TYPE CTR_SIGNALS_INTERNAL :
STRUCT
	//motion control signals
	Enable					:BOOL;
	Execute_SPOS			:BOOL;
	Execute_MABS			:BOOL;
	Execute_MREL			:BOOL;
	Execute_RES				:BOOL;
	//Execute_VEL				:BOOL;
	Execute_HALT			:BOOL;
	Execute_STOP			:BOOL;
	Execute_HOME			:BOOL;	
	JogFw					:BOOL;
	JogBw					:BOOL;
	JogMode					:E_JogMode;
	SetLocation				:LREAL;
	SetPosition				:LREAL;
	SetVelocity				:LREAL;
	SetAccel				:LREAL;
	LimPos					:BOOL;
	LimNeg					:BOOL;
	IsHoming				:BOOL	:= FALSE;
	
	//axis coupling control
	ExecuteCouple			:BOOL; //connected to GearIn
	ExecuteUncouple			:BOOL; //connected to GearOut
	AxisToCouple			:AXIS_REF;
	
	
END_STRUCT
END_TYPE

(* stored: Version 1.1.0.1, ProductVersion 3.1.4026.18
   DUT CTR_SIGNALS_INTERNAL: Id {ce9c7db3-6c6a-44c1-8a13-90802621fe81} *)
